(*~
	<docu>
		<summary>
			Provides standard dialog to interact with the user.		    			 					
 		</summary>
		<example>										
			[!code-pas[StandardDialog](~/../TcOpen/src/TcoInspectors/src/XAE/XAE/TcoInspectorsTests/POUs/Examples/ExampleContext.TcPOU?name=StandardDialog)]		
			[!code-csharp[DialogInitialization](~/../TcOpen/src/TcoInspectors/tests/Sandbox.TcoInspectors.Wpf/App.xaml.cs?name=DialogProxyServiceInitialization)]
		</example>					
	</docu>	
~*)
FUNCTION_BLOCK TcoDialog EXTENDS TcoDialogBase IMPLEMENTS ITcoDialogFormat, ITcoDialogAnswer
VAR
    _text       : STRING(500);
    _caption    : STRING(255);
    _hasOK      : BOOL;
    _hasYes     : BOOL;
    _hasNo      : BOOL;
    _hasCancel  : BOOL;
    _answer     : eDialogAnswer;
    _dialogType : eDialogType;
	_rTrig		: R_TRIG;
	_externalCloseReq : BOOL;
	_closeSignal: BOOL;
END_VAR

SUPER^();

{attribute 'hide'}
{attribute 'obsolete' := 'You should access the property via `ITcoDialogAnswer)` interface.'}
(*~
	<docu>
		<summary>
			Gets the answer from the dialog. 			 					
 		</summary>					
	</docu>	
~*)
PROPERTY Answer : eDialogAnswer
GET
Answer := _answer;
END_GET
END_PROPERTY

{attribute 'hide'}
METHOD PUBLIC FB_init : BOOL
VAR_INPUT
	bInitRetains : BOOL; // if TRUE, the retain variables are initialized (warm start / cold start)
	bInCopyCode : BOOL;  // if TRUE, the instance afterwards gets moved into the copy code (online change)
	ParentObject : ITcoObject;
END_VAR
END_METHOD

METHOD PROTECTED OnStart
SUPER^.OnStart();
_answer := eDialogAnswer.NoAnswer;
END_METHOD

METHOD Restore : ITcoRestorable
VAR_INPUT
END_VAR
SUPER^.Restore();
_externalCloseReq := FALSE;
_closeSignal:=FALSE;
END_METHOD

(*~
	<docu>
		<summary>
			Shows the dialog.
			<note type="important">
				In order for the dialog to be displayed to the user user application must initialized in the user application.
				How to set up the observer in a WPF see `TcOpen.Inxton.TcoCore.Wpf.DialogProxyService`.
			</note> 			 					
 		</summary>					
	</docu>	
~*)
METHOD Show : ITcoDialogFormat
IF THIS^._taskState=eTaskState.Ready THEN
	_answer:=eDialogAnswer.NoAnswer;
END_IF

THIS^.Invoke();
SUPER^();

_hasOK       := FALSE;
_hasYes      := FALSE;
_hasNo       := FALSE;
_hasCancel   := FALSE;
_text        := '';
_caption     := '';
_dialogType  := eDialogType.Undefined;

Show := THIS^;

IF THIS^._taskState=eTaskState.Done AND _answer<>eDialogAnswer.NoAnswer THEN
	THIS^.Restore();
END_IF;
END_METHOD

METHOD ShowWithExternalClose : ITcoDialogFormat
VAR_INPUT
	inCloseSignal:BOOL;
	inDialogAnswerType : eDialogAnswer;

END_VAR
IF THIS^._taskState=eTaskState.Ready THEN
	_answer:=eDialogAnswer.NoAnswer;
END_IF

THIS^.Invoke();
SUPER^();


_hasOK       := FALSE;
_hasYes      := FALSE;
_hasNo       := FALSE;
_hasCancel   := FALSE;
_externalCloseReq := TRUE;
_text        := '';
_caption     := '';
_dialogType  := eDialogType.Undefined;

ShowWithExternalClose := THIS^;
_rTrig(CLK:=inCloseSignal);
IF _rTrig.q THEN
	_closeSignal:=TRUE;
END_IF

IF	_closeSignal THEN
	_answer:=inDialogAnswerType;		
END_IF

IF THIS^._taskState=eTaskState.Done AND _answer<>eDialogAnswer.NoAnswer THEN	
	THIS^.Restore();
END_IF;
END_METHOD

(*~
	<docu>
		<summary>
			Sets the caption of the dialog window. 			 					
 		</summary>					
	</docu>	
~*)
{attribute 'hide'}
{attribute 'obsolete' := 'You should access the method via `Show()` method.'}
METHOD WithCaption : ITcoDialogAnswer
VAR_INPUT
	inCaption : STRING(255);
END_VAR
_caption := inCaption;
WithCaption := THIS^;
END_METHOD

(*~
	<docu>
		<summary>
			Sets that the `OK` button should be available in the dialog prompt. 			 					
 		</summary>					
	</docu>	
~*)
{attribute 'hide'}
{attribute 'obsolete' := 'You should access the method via `Show()` method.'}
METHOD WithOk : ITcoDialogAnswer
VAR_INPUT
END_VAR
_hasOK := TRUE;
WithOk := THIS^;
END_METHOD

(*~
	<docu>
		<summary>
			Sets the text of the dialog window. 			 					
 		</summary>					
	</docu>	
~*)
{attribute 'hide'}
{attribute 'obsolete' := 'You should access the method via `Show()` method.'}
METHOD WithText : ITcoDialogAnswer
VAR_INPUT
	inText : STRING(500);
END_VAR
_text := inText;
WithText := THIS^;
END_METHOD

METHOD WithType : ITcoDialogAnswer
VAR_INPUT
	inDialogType : eDialogType;
END_VAR
_dialogType := inDialogType;
WithType := THIS^;
END_METHOD

(*~
	<docu>
		<summary>
			Sets that the `Yes` and `No` buttons should be available in the dialog prompt. 			 					
 		</summary>					
	</docu>	
~*)
{attribute 'hide'}
{attribute 'obsolete' := 'You should access the method via `Show()` method.'}
METHOD WithYesNo : ITcoDialogAnswer
VAR_INPUT
END_VAR
_hasYes := TRUE;
_hasNo := TRUE;
WithYesNo := THIS^;
END_METHOD

(*~
	<docu>
		<summary>
			Sets that the `Yes`, `No` and `Cancel` buttons should be available in the dialog prompt. 			 					
 		</summary>					
	</docu>	
~*)
{attribute 'hide'}
{attribute 'obsolete' := 'You should access the method via `Show()` method.'}
METHOD WithYesNoCancel : ITcoDialogAnswer
_hasYes    := TRUE;
_hasNo     := TRUE;
_hasCancel := TRUE;
WithYesNoCancel := THIS^;
END_METHOD

END_FUNCTION_BLOCK

(* stored: Version 1.1.0.1
   POU TcoDialog: Id {bc7600eb-cc99-0e0c-2ff6-dcdca22ab5d8}, SpecialFunc None
   Folder Format: Id {b0c49a7f-fe98-0c97-3df9-c74e738844dd}
   Property Answer: Id {0dc2ad34-f12f-0475-2e9e-47acff8b3ab7}
   Get Get: Id {4bbfee3b-9674-0bb1-0d39-17fce0ea4024}
   Method FB_init: Id {155d4d3f-f3ce-0be2-0054-4d5fc2900299}
   Method OnStart: Id {889d908b-4444-0ca3-12c3-2ee5a16d4c25}
   Method Restore: Id {b1b04a3a-6e24-00f0-1f54-b5cc0b7efc8c}
   Method Show: Id {052bdc3b-8ff1-0bbd-0fbb-d25a0348416f}
   Method ShowWithExternalClose: Id {43606d08-c3b6-0424-0c8d-256226f8f48d}
   Method WithCaption: Id {e74b3d9a-c845-0bc5-27de-0a52b6eb9b30}
   Method WithOk: Id {c52dd3cb-da74-062c-2ff2-a375c59030c1}
   Method WithText: Id {b4168086-36a7-0b45-302c-c63e929b4cfa}
   Method WithType: Id {8371ef68-745f-059d-039b-804e722e0a09}
   Method WithYesNo: Id {97fb4a7f-33e1-0bb9-1e9b-67e28ca02e2d}
   Method WithYesNoCancel: Id {366a959f-b453-0846-1871-58dde82bbbb0} *)
